{attribute 'GeneratedUsingTerminal: BK1250-0000-0017'}
{attribute addProperty BoxType "BK1250-0000-0017"}
{attribute addProperty Id "Term_387_KL1002KL1002_BB38DA8F0"}
{attribute addProperty CRC "3295526896"}
{attribute addProperty Size "0"}
TYPE A_0016_BK1250_0000_0017_C46DBFF0 EXTENDS BK1250_AEEC0900 :
STRUCT
	{attribute addProperty Name "Term_387_KL1002"}
	Term_387_KL1002 : KL1002_BB38DA8F;
END_STRUCT
END_TYPE

(* stored: Version 1.2.0.0, ProductVersion 3.1.4024.9
   DUT A_0016_BK1250_0000_0017_C46DBFF0: Id {bc367117-8e56-4219-9014-6020b8b1df9e} *)
